PROGRAM P_Demo_FB_TzSpecificLocalTimeToSystemTime
VAR
    fbFB_TzSpecificLocalTimeToSystemTime : FB_TzSpecificLocalTimeToSystemTime; // FB_TzSpecificLocalTimeToSystemTime 实例
    in                                   : TIMESTRUCT := (wYear:=1970, wMonth:=1, wDay:=1);
    tzInfo                               : ST_TimeZoneInformation;
    out                                  : TIMESTRUCT;
    eTzID                                : E_TimeZoneID;
    bB                                   : BOOL;
END_VAR

// =============================================================================
// 场景：FB_TzSpecificLocalTimeToSystemTime 的最小可编译演示——所有 VAR_INPUT 均以 doc/PDF 中真实引脚名调用。
//       业务侧请在线 monitor / 在线写值触发对应输入，看输出端 monitor 结果。
//
// 价值：保证示例 ST 代码所有引脚名与 FB_TzSpecificLocalTimeToSystemTime 的 VAR_INPUT/VAR_OUTPUT 一致，
//       Add Existing Item (.TcPOU) → 编译 → 登录 流程能跑通，作为 hand-curated 例程
//       的脚手架。
//
// 验证步骤：
//   1. 引用 Tc2_Utilities（及其依赖 Tc2_System）
//   2. 右键 PLC 项目下 POUs 文件夹 → Add → Existing Item → 选本 .TcPOU 文件 → OK → 编译、登录
//   3. 在线对 VAR_INPUT 写入合适触发值（典型 bExecute / RUN / START 上升沿）
//   4. 在线 monitor VAR_OUTPUT 观察 FB 反应
// =============================================================================

fbFB_TzSpecificLocalTimeToSystemTime(
    in := in,
    tzInfo := tzInfo,
    out => out,
    eTzID => eTzID,
    bB => bB
);

END_PROGRAM

(* stored: Version 1.1.0.1, ProductVersion 3.1.4024.5
   POU P_Demo_FB_TzSpecificLocalTimeToSystemTime: Id {dc2044bf-5dfe-5899-a3c1-409b08204dc5}, SpecialFunc None *)
